// TIA Portal V20 export
DATA_BLOCK "PRODUCTION_DATA_HMI_IF_DB"   // DB53
TITLE = HMI und Anwender Schnittstelle für Produktionsdaten / HMI and user interface for production data / HMI 和 用户界面 给 生产 数据
{ S7_Optimized_Access := 'TRUE' }
AUTHOR : Tesla
FAMILY : ProdData
// FUNKTIONSBESCHREIBUNG: 
// Der Baustein beinhaltet alle Informationen zum und vom HMI, sowie die Anwenderschnittstellen für die Produktionsdaten
// Weitere Hinweise: siehe SICAR anwenderdefinierte Dokumentation / SICAR Online-Hilfe.
// DESCRIPTION OF FUNCTIONS:
// 描述 OF 功能:
// stored: MemoryReserve 100
   VAR
      No_DataSets : Struct   // Anzahl konfigurierter Datensätze / Information number of DataSets / 信息 数量 of DataSets
         Limits : Int;
         "Timer" : Int;
         "Counter" : Int;
         ShiftCounter : Int;
      END_STRUCT;
   END_VAR
   VAR RETAIN
      Limit_DataSet : Array[0.."No_of_DataSets_LimitValues"] of Struct   // Datensätze Grenzwerte / DataSets Limit value / DataSets 限制 值
         Enabled : Array[0..10] of Bool;
         Remainder_Value : Array[0..16] of UInt;   // Restwert / Remainder value / Remainder 值
         Set_Point_Value : Array[0..16] of UInt;   // Sollwert / SetPoint value / 设定点 值
         Prewarn_Value : Array[0..16] of UInt;   // Vorwarnsollwert / Prewarn value / Prewarn 值
         Control { ExternalAccessible := 'False'; ExternalVisible := 'False'; ExternalWritable := 'False'; S7_SetPoint := 'True'} : Array[0..16] of "LIMIT_VALUE_CTRL_UDT";   // Steuerung / Control / 控制
         "ColorCode_Alarm/Prewarn" : Array[0..16] of UInt;   // Farbcode für Alarm/Vorwarnung / ColorCode Alarm/Prewarn / ColorCode 警报/Prewarn
         ColorCode_SelectButton : UInt;   // Farbcode für Auswahl Button / ColorCode selcect-button / ColorCode selcect-按钮
         Index_selected_Counter : UInt;   // Index gewählter Zähler zum Löschen / Index selected counter for reset from HMI / Index 选择的 计数器 给 重置 从 HMI
         DivButton : Byte;   // %0=Reset / %0=重置
      END_STRUCT;
   END_VAR
   VAR
      ColorCode_SelectButton : Array[0..8] of UInt;   // Farbcode für Datensatz Anwahl Button / ColorCode for data set select button / ColorCode 给 数据 设置 选择 按钮
   END_VAR
   VAR RETAIN
      CycleTimer_DataSet : Array[0.."No_of_DataSets_CycleTimer"] of Struct   // Datensätze Taktzeiten / DataSets Cycle timer / DataSets 周期 记时器
         Enabled : Array[0..20] of Bool;
         Timer_Value : Array[0..20] of UInt;   // Messwerte / Measured value / 测量的 值
         Timer_Average_Value : Array[0..20] of UInt;   // Mittelwert Messwerte / Average of measurement values / 平均 of 测量 值
         Number_of_Counts : Array[0..20] of UInt;   // Anzahl Messungen für Mittelwerte / Number of measurements for average values / 数量 of measurements 给 平均 值
         Timer_Target_Value : Array[0..20] of UInt;   // Sollwerte / Set values / 设置 值
         Measurement_active : Array[0..20] of Bool;   // Messung aktiv / Measurement active / 测量 现行
         Index_selected_Timer : UInt;   // Index angewählter Wert zum Löschen / Index selected value to be cleared / Index 选择的 值 到 be cleared
         DivButton : Byte;   // %X0=Reset Average einzel, %X1=Reset Average All / %X0=Reset Average single, %X1=Reset Average All / %X0=重置 平均 单, %X1=重置 平均 全部
         Control { ExternalAccessible := 'False'; ExternalVisible := 'False'; ExternalWritable := 'False'; S7_SetPoint := 'True'} : Array[0..20] of "CYCLE_TIMER_CTRL_UDT";   // Anwender-Schnittstelle Taktzeiten / User interface cycle times / 用户界面 周期 times
         Reset_Average_All_ext { ExternalAccessible := 'False'; ExternalVisible := 'False'; ExternalWritable := 'False'} : Bool;   // Anwender-Schnittstelle löschen Mittelwerte / User interface clear averages / 用户界面 清除 averages
      END_STRUCT;
      Counter_DataSet : Array[0.."No_of_DataSets_Counter"] of Struct   // Datensätze Zähler / DataSets Counter / DataSets 计数器
         Enabled : Array[0..20] of Bool;
         Counter_Value : Array[0..20] of UInt;
         Control { ExternalAccessible := 'False'; ExternalVisible := 'False'; ExternalWritable := 'False'; S7_SetPoint := 'True'} : Array[0..20] of "COUNTER_CTRL_UDT";
         Reset_All_ext { ExternalAccessible := 'False'; ExternalVisible := 'False'; ExternalWritable := 'False'} : Bool;
         Index_selected_Counter : UInt;
         DivButton : Byte;   // %X0=Reset einzel, %X1=ResetAll / %X0=Reset single, %X1=ResetAll / %X0=重置 单, %X1=ResetAll
      END_STRUCT;
      ShiftCounter_DataSet : Array[0.."No_of_DataSets_ShiftCounter"] of Struct   // Datensätze Schichtzähler / DataSets ShiftCounter / DataSets 工作轮班记数器
         Enabled : Array[0..10] of Bool;   // Tesla addition: must set high to enable shift counter / Tesla addition: 必须 设置 high 到 启用 工作轮班 计数器
         ShiftCounter_CurrentValue : Array[0..10] of UInt;
         ShiftCounter_CurrentTarget : Array[0..10] of UInt;
         ShiftCounter_PreviousValue : Array[0..10] of UInt;
         ShiftCounter_PreviousTarget : Array[0..10] of UInt;
         ShiftCounter_PenultimateValue : Array[0..10] of UInt;
         ShiftCounter_PenultimateTarget : Array[0..10] of UInt;
         Control { ExternalAccessible := 'False'; ExternalVisible := 'False'; ExternalWritable := 'False'} : Array[0..10] of Bool;
         Reset_All_ext { ExternalAccessible := 'False'; ExternalVisible := 'False'; ExternalWritable := 'False'} : Bool;
         DivButton : Byte;   // %0=ResetAll
      END_STRUCT;
      ProductionRecord : Struct
         DTL : DTL;
         "DT" : Date_And_Time;
         Retval : Int;
         StartTime : Array[1..7] of Date_And_Time;
         StopTime : Array[1..7] of Date_And_Time;
         Count : Array[1..7] of UInt;
         Start : Bool;
         Stop : Bool;
         Reset : Bool;
         StartIndicate : Bool;
         StopIndicate : Bool;
         ONS1 : Bool;
         ONS2 : Bool;
         Start_Delay : Struct
            temp : Bool;
            transfout_tm : Bool;
            start : Bool;
         END_STRUCT;
      END_STRUCT;
   END_VAR
BEGIN
   CycleTimer_DataSet[1].Timer_Average_Value[2] := 0;
END_DATA_BLOCK
